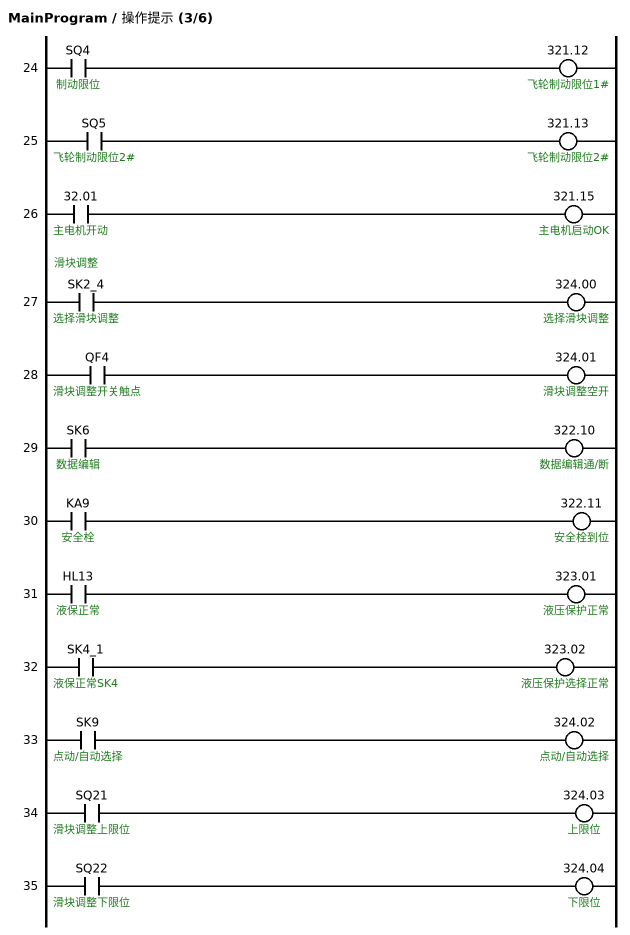
; [picture p48: MainProgram / 操作提示, rungs 24-35]
; rung 24
LD SQ4  ; 制动限位
OUT 321.12  ; 飞轮制动限位1#
; rung 25
LD SQ5  ; 飞轮制动限位2#
OUT 321.13  ; 飞轮制动限位2#
; rung 26
LD 32.01  ; 主电机开动
OUT 321.15  ; 主电机启动OK
; rung 27: 滑块调整
LD SK2_4  ; 选择滑块调整
OUT 324.00  ; 选择滑块调整
; rung 28
LD QF4  ; 滑块调整开关触点
OUT 324.01  ; 滑块调整空开
; rung 29
LD SK6  ; 数据编辑
OUT 322.10  ; 数据编辑通/断
; rung 30
LD KA9  ; 安全栓
OUT 322.11  ; 安全栓到位
; rung 31
LD HL13  ; 液保正常
OUT 323.01  ; 液压保护正常
; rung 32
LD SK4_1  ; 液保正常SK4
OUT 323.02  ; 液压保护选择正常
; rung 33
LD SK9  ; 点动/自动选择
OUT 324.02  ; 点动/自动选择
; rung 34
LD SQ21  ; 滑块调整上限位
OUT 324.03  ; 上限位
; rung 35
LD SQ22  ; 滑块调整下限位
OUT 324.04  ; 下限位

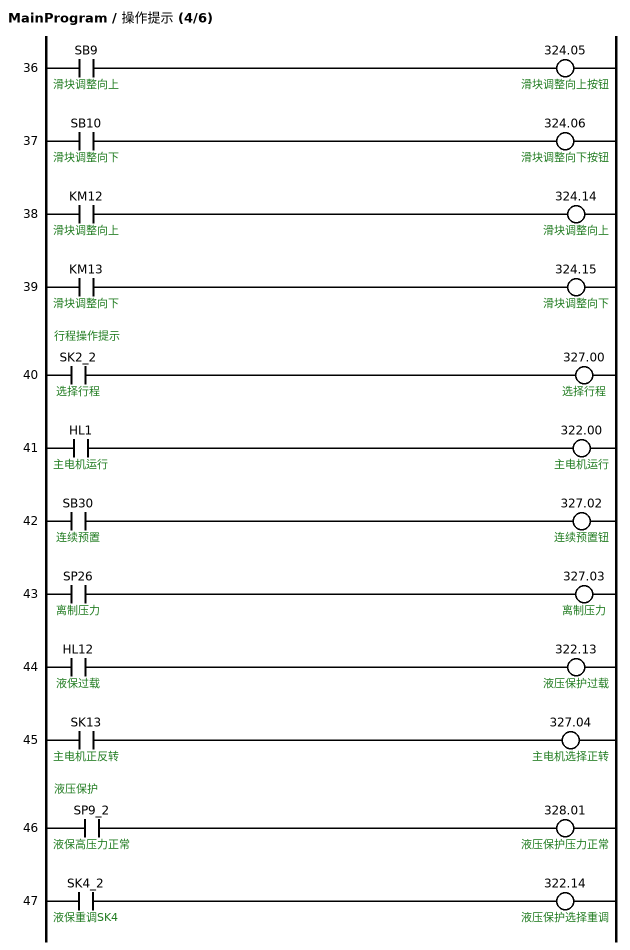
; rung 36
LD SB9  ; 滑块调整向上
OUT 324.05  ; 滑块调整向上按钮
; rung 37
LD SB10  ; 滑块调整向下
OUT 324.06  ; 滑块调整向下按钮
; rung 38
LD KM12  ; 滑块调整向上
OUT 324.14  ; 滑块调整向上
; rung 39
LD KM13  ; 滑块调整向下
OUT 324.15  ; 滑块调整向下
; rung 40: 行程操作提示
LD SK2_2  ; 选择行程
OUT 327.00  ; 选择行程
; rung 41
LD HL1  ; 主电机运行
OUT 322.00  ; 主电机运行
; rung 42
LD SB30  ; 连续预置
OUT 327.02  ; 连续预置钮
; rung 43
LD SP26  ; 离制压力
OUT 327.03  ; 离制压力
; rung 44
LD HL12  ; 液保过载
OUT 322.13  ; 液压保护过载
; rung 45
LD SK13  ; 主电机正反转
OUT 327.04  ; 主电机选择正转
; rung 46: 液压保护
LD SP9_2  ; 液保高压力正常
OUT 328.01  ; 液压保护压力正常
; rung 47
LD SK4_2  ; 液保重调SK4
OUT 322.14  ; 液压保护选择重调

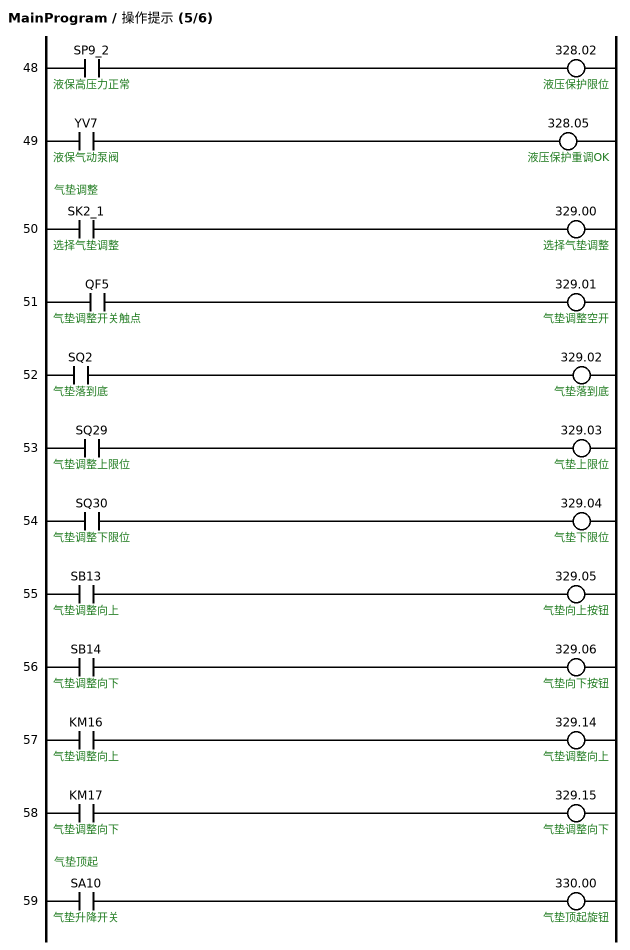
; rung 48
LD SP9_2  ; 液保高压力正常
OUT 328.02  ; 液压保护限位
; rung 49
LD YV7  ; 液保气动泵阀
OUT 328.05  ; 液压保护重调OK
; rung 50: 气垫调整
LD SK2_1  ; 选择气垫调整
OUT 329.00  ; 选择气垫调整
; rung 51
LD QF5  ; 气垫调整开关触点
OUT 329.01  ; 气垫调整空开
; rung 52
LD SQ2  ; 气垫落到底
OUT 329.02  ; 气垫落到底
; rung 53
LD SQ29  ; 气垫调整上限位
OUT 329.03  ; 气垫上限位
; rung 54
LD SQ30  ; 气垫调整下限位
OUT 329.04  ; 气垫下限位
; rung 55
LD SB13  ; 气垫调整向上
OUT 329.05  ; 气垫向上按钮
; rung 56
LD SB14  ; 气垫调整向下
OUT 329.06  ; 气垫向下按钮
; rung 57
LD KM16  ; 气垫调整向上
OUT 329.14  ; 气垫调整向上
; rung 58
LD KM17  ; 气垫调整向下
OUT 329.15  ; 气垫调整向下
; rung 59: 气垫顶起
LD SA10  ; 气垫升降开关
OUT 330.00  ; 气垫顶起旋钮

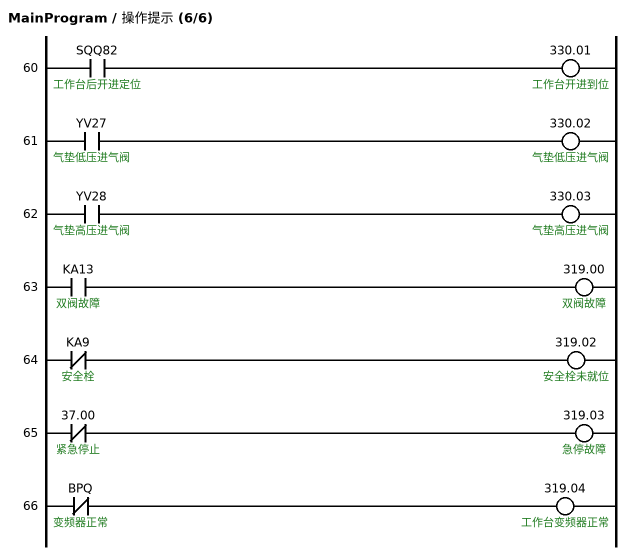
; rung 60
LD SQQ82  ; 工作台后开进定位
OUT 330.01  ; 工作台开进到位
; rung 61
LD YV27  ; 气垫低压进气阀
OUT 330.02  ; 气垫低压进气阀
; rung 62
LD YV28  ; 气垫高压进气阀
OUT 330.03  ; 气垫高压进气阀
; rung 63
LD KA13  ; 双阀故障
OUT 319.00  ; 双阀故障
; rung 64
LDNOT KA9  ; 安全栓
OUT 319.02  ; 安全栓未就位
; rung 65
LDNOT 37.00  ; 紧急停止
OUT 319.03  ; 急停故障
; rung 66
LDNOT BPQ  ; 变频器正常
OUT 319.04  ; 工作台变频器正常

### Section 模具夹紧

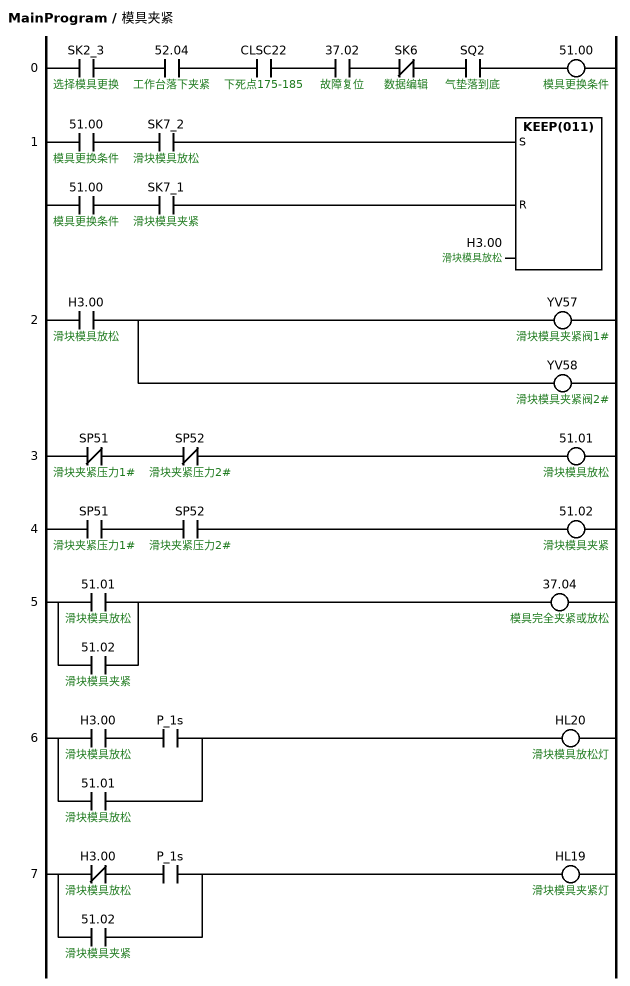
; rung 0
LD SK2_3  ; 选择模具更换
AND 52.04  ; 工作台落下夹紧
AND CLSC22  ; 下死点175-185
AND 37.02  ; 故障复位
ANDNOT SK6  ; 数据编辑
AND SQ2  ; 气垫落到底
OUT 51.00  ; 模具更换条件
; rung 1
LD 51.00  ; 模具更换条件
AND SK7_2  ; 滑块模具放松
LD 51.00  ; 模具更换条件
AND SK7_1  ; 滑块模具夹紧
KEEP(011) H3.00  ; 滑块模具放松
; rung 2
LD H3.00  ; 滑块模具放松
OUT YV57  ; 滑块模具夹紧阀1#
OUT YV58  ; 滑块模具夹紧阀2#
; rung 3
LDNOT SP51  ; 滑块夹紧压力1#
ANDNOT SP52  ; 滑块夹紧压力2#
OUT 51.01  ; 滑块模具放松
; rung 4
LD SP51  ; 滑块夹紧压力1#
AND SP52  ; 滑块夹紧压力2#
OUT 51.02  ; 滑块模具夹紧
; rung 5
LD 51.01  ; 滑块模具放松
OR 51.02  ; 滑块模具夹紧
OUT 37.04  ; 模具完全夹紧或放松
; rung 6
LD H3.00  ; 滑块模具放松
AND P_1s
OR 51.01  ; 滑块模具放松
OUT HL20  ; 滑块模具放松灯
; rung 7
LDNOT H3.00  ; 滑块模具放松
AND P_1s
OR 51.02  ; 滑块模具夹紧
OUT HL19  ; 滑块模具夹紧灯

### Section END
; rung 0
END(001)